{attribute addProperty BoxType "EJ7037-0000-0020"}
{attribute addProperty Id "StatusAT %I*Status_E26627ED1621Counter_valueAT %I*UINT16217Latch_valueAT %I*UINT16218"}
{attribute addProperty CRC "3666293612"}
{attribute addProperty SizeInBites "48"}
{attribute addProperty SizeInBytes "6"}
TYPE ENC_Status_compact_DA87336C :
STRUCT
	{attribute addProperty Name "Status"}
	Status AT %I* : Status_E26627ED;
	{attribute addProperty Name "Counter_value"}
	Counter_value AT %I* : UINT;
	{attribute addProperty Name "Latch_value"}
	Latch_value AT %I* : UINT;
END_STRUCT
END_TYPE

(* stored: Version 1.2.0.0, ProductVersion 3.1.4024.9
   DUT ENC_Status_compact_DA87336C: Id {dcbbb6aa-c4bb-47de-9969-4c8cba98f00e} *)
